INTERFACE IEventHandler_OnSecondsChanged EXTENDS IEventHandlerBase

METHOD OnSecondsChanged
VAR_INPUT
	Now: TIMESTRUCT;
END_VAR
END_METHOD

END_INTERFACE

(* stored: Version 1.1.0.1, ProductVersion 3.1.4024.3
   Itf IEventHandler_OnSecondsChanged: Id {e93a60ca-2df2-098f-3bcc-523bc3075eca}
   Method OnSecondsChanged: Id {f5e672c0-5719-0faa-26fb-44b840e26d02} *)
